TYPE ST_MotionlinxAI_Controller_Command :
	STRUCT
		Extend	: BOOL;
		Retract : BOOL;
	END_STRUCT
END_TYPE

(* stored: Version 1.1.0.1, ProductVersion 3.1.4024.15
   DUT ST_MotionlinxAI_Controller_Command: Id {11cf0a91-77c2-4131-8626-b12a72606b35} *)
